FUNCTION_BLOCK FB_ValveControl (* Basic Function Block Type *)
  (* Standard: 61499-2 *)
  (* Version 0.0, 2014-5-4, wildai, nxtControl GmbH, Template *)
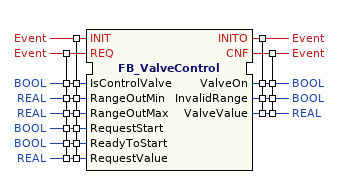
  EVENT_INPUT
    INIT WITH IsControlValve, RangeOutMin, RangeOutMax, RequestStart, ReadyToStart, RequestValue; (* Initialization Request *)
    REQ WITH IsControlValve, RangeOutMin, RangeOutMax, RequestStart, ReadyToStart, RequestValue; (* Normal Execution Request *)
  END_EVENT
  EVENT_OUTPUT
    INITO WITH ValveOn, InvalidRange, ValveValue; (* Initialization Confirm *)
    CNF WITH ValveOn, InvalidRange, ValveValue; (* Execution Confirmation *)
  END_EVENT
  VAR_INPUT
    IsControlValve : BOOL; (* Input event qualifier *)
    RangeOutMin : REAL;
    RangeOutMax : REAL;
    RequestStart : BOOL;
    ReadyToStart : BOOL;
    RequestValue : REAL;
  END_VAR
  VAR_OUTPUT
    ValveOn : BOOL; (* Output event qualifier *)
    InvalidRange : BOOL;
    ValveValue : REAL;
  END_VAR
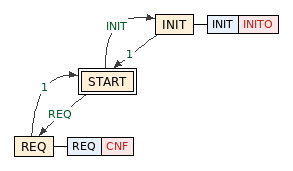
  EC_STATES
    START; (* Initial State *)
    INIT : INIT -> INITO; (* Initialization *)
    REQ : REQ -> CNF; (* Normal execution *)
  END_STATES
  EC_TRANSITIONS
    START TO INIT := INIT;
    INIT TO START := 1;
    START TO REQ := REQ;
    REQ TO START := 1;
  END_TRANSITIONS
  ALGORITHM INIT IN ST: (* Initialization algorithm *)
;

ValveOn := FALSE;
InvalidRange := FALSE;
ValveValue := 0.0;
  END_ALGORITHM
  ALGORITHM REQ IN ST: (* Normally executed algorithm *)
;

IF IsControlValve AND RequestStart AND ReadyToStart THEN
	IF RequestValue >= RangeOutMin AND RequestValue <= RangeOutMax THEN
		ValveValue := RequestValue;
		InvalidRange := FALSE;
		ValveOn := TRUE;
	ELSE
		ValveValue := 0.0;
		InvalidRange := TRUE;
		ValveOn := FALSE;
	END_IF;
ELSE
	ValveOn := FALSE;
	ValveValue := 0.0;
END_IF;
  END_ALGORITHM
END_FUNCTION_BLOCK
